(* CODESYS project Codesys

Project tree, tasks and I/O mapping:
  Device : PMCprimo Base, Pilz GmbH & Co. KG, version 3.5.15.1
    application Application
      libraries: Standard, 3.5.18.0 (System)
      task EtherCAT (externalevent, external event EVENT_ECM_DC, priority 0) calls EtherCAT_Master_Pilz.EtherCAT_Task, PLC_PRG
      task MainTask (cyclic, interval 1 ms, priority 0) calls nothing
      program PLC_PRG [LD]
    EtherCAT_Master_Pilz : EtherCAT_Master_Pilz, Pilz GmbH & Co. KG, version 3.5.17.0
        settings: NetworkName = 'ETHERCAT'; NetworkName = "ETHERCAT"; SrcAddress1 = 2; SrcAddress2 = 1212745857
      SI6_SC6_2Ax : SI6/SC6 2Ax, STOEBER ANTRIEBSTECHNIK GmbH & Co. KG, order no. SI6/SC6 2Ax, version Revision=16#00000011
          settings: ModularDevice = True; Number of Outputs = 0; Number of Inputs = 0; Number of Infos about Outputs = 0; Number of Infos about Inputs = 0; MDP_InputOffsets = [0,0,192]; MDP_OutputOffsets = [0,0,48]; Sync.Length = 12; Sync.Length = 44; FMMU.Length = 12; FMMU.Length = 44; Number of RxPDOs of the Slave = 2; Number of TxPDOs of the Slave = 2; DC sync0 cycletime = 1000; DC sync1 cycletime = 1000; RxTxPdo.NumberofExcludes = 0; RxTxPdo.NumberofEntries = 2; RxTxPdo.Index = 16#1600; RxTxPdo.Fixed = False; RxTxPdo.Mandatory = False; RxTxPdo.Virtual = False; RxTxPdo.Sm = 2; RxTxPdo.Su = 0; RxTxPdo.Name = 'Axis A to Slave'; RxTxPdo.DependOnSlot = False; RxTxPdo.DependOnSlotGroup = False; RxTxPdo.OverwrittenByModule = True; 1.A515 Controlword.Index = 16#6040; 1.A515 Controlword.SubIndex = 0; 1.A515 Controlword.Size = 16; 1.A515 Controlword.Offset = 0; 1.A515 Controlword.DependOnSlot = False; 1.A515 Controlword.DependOnSlotGroup = False; 1.A567 Target position.Index = 16#607A; 1.A567 Target position.SubIndex = 0; 1.A567 Target position.Size = 32; 1.A567 Target position.Offset = 0; 1.A567 Target position.DependOnSlot = False; 1.A567 Target position.DependOnSlotGroup = False; RxTxPdo.NumberofExcludes = 0;
            RxTxPdo.NumberofEntries = 2; RxTxPdo.Index = 16#1601; RxTxPdo.Fixed = False; RxTxPdo.Mandatory = False; RxTxPdo.Virtual = False; RxTxPdo.Sm = 2; RxTxPdo.Su = 0; RxTxPdo.Name = 'Axis B to Slave'; RxTxPdo.DependOnSlot = False; RxTxPdo.DependOnSlotGroup = False; RxTxPdo.OverwrittenByModule = True; 2.A515 Controlword.Index = 16#6840; 2.A515 Controlword.SubIndex = 0; 2.A515 Controlword.Size = 16; 2.A515 Controlword.Offset = 0; 2.A515 Controlword.DependOnSlot = False; 2.A515 Controlword.DependOnSlotGroup = False; 2.A567 Target position.Index = 16#687A; 2.A567 Target position.SubIndex = 0; 2.A567 Target position.Size = 32; 2.A567 Target position.Offset = 0; 2.A567 Target position.DependOnSlot = False; 2.A567 Target position.DependOnSlotGroup = False; RxTxPdo.NumberofExcludes = 0; RxTxPdo.NumberofEntries = 8; RxTxPdo.Index = 16#1A00; RxTxPdo.Fixed = False; RxTxPdo.Mandatory = False; RxTxPdo.Virtual = False; RxTxPdo.Sm = 3; RxTxPdo.Su = 0; RxTxPdo.Name = 'Axis A to Master'; RxTxPdo.DependOnSlot = False; RxTxPdo.DependOnSlotGroup = False; RxTxPdo.OverwrittenByModule = True; 1.A516 Statusword.Index = 16#6041; 1.A516 Statusword.SubIndex = 0; 1.A516 Statusword.Size = 16; 1.A516 Statusword.Offset = 0; 1.A516 Statusword.DependOnSlot = False;
            1.A516 Statusword.DependOnSlotGroup = False; 1.A545 Position actual value.Index = 16#6064; 1.A545 Position actual value.SubIndex = 0; 1.A545 Position actual value.Size = 32; 1.A545 Position actual value.Offset = 0; 1.A545 Position actual value.DependOnSlot = False; 1.A545 Position actual value.DependOnSlotGroup = False; 1.A564 Torque actual value.Index = 16#6077; 1.A564 Torque actual value.SubIndex = 0; 1.A564 Torque actual value.Size = 16; 1.A564 Torque actual value.Offset = 0; 1.A564 Torque actual value.DependOnSlot = False; 1.A564 Torque actual value.DependOnSlotGroup = False; 1.A636 Digital inputs.Index = 16#60FD; 1.A636 Digital inputs.SubIndex = 0; 1.A636 Digital inputs.Size = 32; 1.A636 Digital inputs.Offset = 0; 1.A636 Digital inputs.DependOnSlot = False; 1.A636 Digital inputs.DependOnSlotGroup = False; 1.A595 Touch probe status.Index = 16#60B9; 1.A595 Touch probe status.SubIndex = 0; 1.A595 Touch probe status.Size = 16; 1.A595 Touch probe status.Offset = 0; 1.A595 Touch probe status.DependOnSlot = False; 1.A595 Touch probe status.DependOnSlotGroup = False; 1.A596 Touch probe position 1 positive value.Index = 16#60BA; 1.A596 Touch probe position 1 positive value.SubIndex = 0; 1.A596 Touch probe position 1 positive value.Size = 32; 1.A596 Touch probe position 1 positive value.Offset = 0; 1.A596 Touch probe position 1 positive value.DependOnSlot = False; 1.A596 Touch probe position 1 positive value.DependOnSlotGroup = False; 1.A597 Touch probe position 1 negative value.Index = 16#60BB; 1.A597 Touch probe position 1 negative value.SubIndex = 0; 1.A597 Touch probe position 1 negative value.Size = 32; 1.A597 Touch probe position 1 negative value.Offset = 0; 1.A597 Touch probe position 1 negative value.DependOnSlot = False; 1.A597 Touch probe position 1 negative value.DependOnSlotGroup = False; 1.E201 Statuswort 2.Index = 16#28C9; 1.E201 Statuswort 2.SubIndex = 0; 1.E201 Statuswort 2.Size = 16;
            1.E201 Statuswort 2.Offset = 0; 1.E201 Statuswort 2.DependOnSlot = False; 1.E201 Statuswort 2.DependOnSlotGroup = False; RxTxPdo.NumberofExcludes = 0; RxTxPdo.NumberofEntries = 7; RxTxPdo.Index = 16#1A01; RxTxPdo.Fixed = False; RxTxPdo.Mandatory = False; RxTxPdo.Virtual = False; RxTxPdo.Sm = 3; RxTxPdo.Su = 0; RxTxPdo.Name = 'Axis B to Master'; RxTxPdo.DependOnSlot = False; RxTxPdo.DependOnSlotGroup = False; RxTxPdo.OverwrittenByModule = True; 2.A516 Statusword.Index = 16#6841; 2.A516 Statusword.SubIndex = 0; 2.A516 Statusword.Size = 16; 2.A516 Statusword.Offset = 0; 2.A516 Statusword.DependOnSlot = False; 2.A516 Statusword.DependOnSlotGroup = False; 2.A545 Position actual value.Index = 16#6864; 2.A545 Position actual value.SubIndex = 0; 2.A545 Position actual value.Size = 32; 2.A545 Position actual value.Offset = 0; 2.A545 Position actual value.DependOnSlot = False; 2.A545 Position actual value.DependOnSlotGroup = False; 2.A564 Torque actual value.Index = 16#6877; 2.A564 Torque actual value.SubIndex = 0; 2.A564 Torque actual value.Size = 16; 2.A564 Torque actual value.Offset = 0; 2.A564 Torque actual value.DependOnSlot = False; 2.A564 Torque actual value.DependOnSlotGroup = False; 2.A595 Touch probe status.Index = 16#68B9; 2.A595 Touch probe status.SubIndex = 0; 2.A595 Touch probe status.Size = 16; 2.A595 Touch probe status.Offset = 0; 2.A595 Touch probe status.DependOnSlot = False; 2.A595 Touch probe status.DependOnSlotGroup = False; 2.A596 Touch probe position 1 positive value.Index = 16#68BA;
            2.A596 Touch probe position 1 positive value.SubIndex = 0; 2.A596 Touch probe position 1 positive value.Size = 32; 2.A596 Touch probe position 1 positive value.Offset = 0; 2.A596 Touch probe position 1 positive value.DependOnSlot = False; 2.A596 Touch probe position 1 positive value.DependOnSlotGroup = False; 2.A597 Touch probe position 1 negative value.Index = 16#68BB; 2.A597 Touch probe position 1 negative value.SubIndex = 0; 2.A597 Touch probe position 1 negative value.Size = 32; 2.A597 Touch probe position 1 negative value.Offset = 0; 2.A597 Touch probe position 1 negative value.DependOnSlot = False; 2.A597 Touch probe position 1 negative value.DependOnSlotGroup = False; 1.E201 Statuswort 2.Index = 16#28C9; 1.E201 Statuswort 2.SubIndex = 0; 1.E201 Statuswort 2.Size = 16; 1.E201 Statuswort 2.Offset = 0; 1.E201 Statuswort 2.DependOnSlot = False; 1.E201 Statuswort 2.DependOnSlotGroup = False; 1.A515 Controlword.Name = '1.A515 Controlword'; 1.A515 Controlword.DataType = 'WORD'; 1.A515 Controlword.Default = ''; 1.A515 Controlword.Comment = ''; 1.A567 Target position.Name = '1.A567 Target position'; 1.A567 Target position.DataType = 'DINT'; 1.A567 Target position.Default = ''; 1.A567 Target position.Comment = ''; 2.A515 Controlword.Name = '2.A515 Controlword'; 2.A515 Controlword.DataType = 'WORD'; 2.A515 Controlword.Default = ''; 2.A515 Controlword.Comment = ''; 2.A567 Target position.Name = '2.A567 Target position'; 2.A567 Target position.DataType = 'DINT'; 2.A567 Target position.Default = ''; 2.A567 Target position.Comment = ''; 1.A516 Statusword.Name = '1.A516 Statusword'; 1.A516 Statusword.DataType = 'WORD'; 1.A516 Statusword.Default = ''; 1.A516 Statusword.Comment = ''; 1.A545 Position actual value.Name = '1.A545 Position actual value'; 1.A545 Position actual value.DataType = 'DINT'; 1.A545 Position actual value.Default = '';
            1.A545 Position actual value.Comment = ''; 1.A564 Torque actual value.Name = '1.A564 Torque actual value'; 1.A564 Torque actual value.DataType = 'INT'; 1.A564 Torque actual value.Default = ''; 1.A564 Torque actual value.Comment = ''; 1.A636 Digital inputs.Name = '1.A636 Digital inputs'; 1.A636 Digital inputs.DataType = 'DWORD'; 1.A636 Digital inputs.Default = ''; 1.A636 Digital inputs.Comment = ''; 1.A595 Touch probe status.Name = '1.A595 Touch probe status'; 1.A595 Touch probe status.DataType = 'WORD'; 1.A595 Touch probe status.Default = ''; 1.A595 Touch probe status.Comment = ''; 1.A596 Touch probe position 1 positive value.Name = '1.A596 Touch probe position 1 positive value'; 1.A596 Touch probe position 1 positive value.DataType = 'DINT'; 1.A596 Touch probe position 1 positive value.Default = ''; 1.A596 Touch probe position 1 positive value.Comment = ''; 1.A597 Touch probe position 1 negative value.Name = '1.A597 Touch probe position 1 negative value'; 1.A597 Touch probe position 1 negative value.DataType = 'DINT'; 1.A597 Touch probe position 1 negative value.Default = ''; 1.A597 Touch probe position 1 negative value.Comment = ''; 1.E201 Statuswort 2.Name = '1.E201 Statuswort 2'; 1.E201 Statuswort 2.DataType = 'WORD'; 1.E201 Statuswort 2.Default = ''; 1.E201 Statuswort 2.Comment = ''; 2.A516 Statusword.Name = '2.A516 Statusword'; 2.A516 Statusword.DataType = 'WORD'; 2.A516 Statusword.Default = ''; 2.A516 Statusword.Comment = ''; 2.A545 Position actual value.Name = '2.A545 Position actual value'; 2.A545 Position actual value.DataType = 'DINT'; 2.A545 Position actual value.Default = ''; 2.A545 Position actual value.Comment = ''; 2.A564 Torque actual value.Name = '2.A564 Torque actual value'; 2.A564 Torque actual value.DataType = 'INT'; 2.A564 Torque actual value.Default = ''; 2.A564 Torque actual value.Comment = ''; 2.A595 Touch probe status.Name = '2.A595 Touch probe status'; 2.A595 Touch probe status.DataType = 'WORD'; 2.A595 Touch probe status.Default = '';
            2.A595 Touch probe status.Comment = ''; 2.A596 Touch probe position 1 positive value.Name = '2.A596 Touch probe position 1 positive value'; 2.A596 Touch probe position 1 positive value.DataType = 'DINT'; 2.A596 Touch probe position 1 positive value.Default = ''; 2.A596 Touch probe position 1 positive value.Comment = ''; 2.A597 Touch probe position 1 negative value.Name = '2.A597 Touch probe position 1 negative value'; 2.A597 Touch probe position 1 negative value.DataType = 'DINT'; 2.A597 Touch probe position 1 negative value.Default = ''; 2.A597 Touch probe position 1 negative value.Comment = ''; 1.E201 Statuswort 2.Name = '1.E201 Statuswort 2'; 1.E201 Statuswort 2.DataType = 'WORD'; 1.E201 Statuswort 2.Default = ''; 1.E201 Statuswort 2.Comment = ''
        Axis_A : xA PMCprimo-SI6/SC6_0, STOEBER ANTRIEBSTECHNIK GmbH & Co. KG, order no. PMCprimo-SI6/SC6_0, version 0
            settings: Number of Outputs = 2; Number of Inputs = 8; Number of Infos about Outputs = 2; Number of Infos about Inputs = 8; RxTxPdo.Mandatory = False; RxTxPdo.Virtual = False; RxTxPdo.DependOnSlot = False; RxTxPdo.DependOnSlotGroup = False; RxTxPdo.OverwrittenByModule = True; 1.A515 Controlword.Offset = 0; 1.A515 Controlword.DependOnSlot = False; 1.A515 Controlword.DependOnSlotGroup = False; 1.A567 Target position.Offset = 0; 1.A567 Target position.DependOnSlot = False; 1.A567 Target position.DependOnSlotGroup = False; RxTxPdo.Mandatory = False; RxTxPdo.Virtual = False; RxTxPdo.DependOnSlot = False; RxTxPdo.DependOnSlotGroup = False; RxTxPdo.OverwrittenByModule = True; 1.A516 Statusword.Offset = 0; 1.A516 Statusword.DependOnSlot = False; 1.A516 Statusword.DependOnSlotGroup = False; 1.A545 Position actual value.Offset = 0; 1.A545 Position actual value.DependOnSlot = False; 1.A545 Position actual value.DependOnSlotGroup = False; 1.A564 Torque actual value.Offset = 0; 1.A564 Torque actual value.DependOnSlot = False; 1.A564 Torque actual value.DependOnSlotGroup = False; 1.A636 Digital inputs.Offset = 0; 1.A636 Digital inputs.DependOnSlot = False; 1.A636 Digital inputs.DependOnSlotGroup = False; 1.A595 Touch probe status.Offset = 0; 1.A595 Touch probe status.DependOnSlot = False; 1.A595 Touch probe status.DependOnSlotGroup = False; 1.A596 Touch probe position 1 positive value.Offset = 0; 1.A596 Touch probe position 1 positive value.DependOnSlot = False; 1.A596 Touch probe position 1 positive value.DependOnSlotGroup = False; 1.A597 Touch probe position 1 negative value.Offset = 0; 1.A597 Touch probe position 1 negative value.DependOnSlot = False;
              1.A597 Touch probe position 1 negative value.DependOnSlotGroup = False; 1.E201 Statuswort 2.Offset = 0; 1.E201 Statuswort 2.DependOnSlot = False; 1.E201 Statuswort 2.DependOnSlotGroup = False; 1.A515 Controlword.Default = ''; 1.A567 Target position.Default = ''; 1.A516 Statusword.Default = ''; 1.A545 Position actual value.Default = ''; 1.A564 Torque actual value.Default = ''; 1.A636 Digital inputs.Default = ''; 1.A595 Touch probe status.Default = ''; 1.A596 Touch probe position 1 positive value.Default = ''; 1.A597 Touch probe position 1 negative value.Default = ''; 1.E201 Statuswort 2.Default = ''
            unmapped channels: 1.A515 Controlword, 1.A567 Target position, 1.A516 Statusword, 1.A545 Position actual value, 1.A564 Torque actual value, 1.A636 Digital inputs, 1.A595 Touch probe status, 1.A596 Touch probe position 1 positive value, 1.A597 Touch probe position 1 negative value, 1.E201 Statuswort 2
        Axis_B : xB PMCprimo-SI6/SC6_1, STOEBER ANTRIEBSTECHNIK GmbH & Co. KG, order no. PMC-SI6/SC6_1, version 0
            settings: Number of Outputs = 2; Number of Inputs = 7; Number of Infos about Outputs = 2; Number of Infos about Inputs = 7; RxTxPdo.Mandatory = False; RxTxPdo.Virtual = False; RxTxPdo.DependOnSlot = False; RxTxPdo.DependOnSlotGroup = False; RxTxPdo.OverwrittenByModule = True; 2.A515 Controlword.Offset = 0; 2.A515 Controlword.DependOnSlot = False; 2.A515 Controlword.DependOnSlotGroup = False; 2.A567 Target position.Offset = 0; 2.A567 Target position.DependOnSlot = False; 2.A567 Target position.DependOnSlotGroup = False; RxTxPdo.Mandatory = False; RxTxPdo.Virtual = False; RxTxPdo.DependOnSlot = False; RxTxPdo.DependOnSlotGroup = False; RxTxPdo.OverwrittenByModule = True; 2.A516 Statusword.Offset = 0; 2.A516 Statusword.DependOnSlot = False; 2.A516 Statusword.DependOnSlotGroup = False; 2.A545 Position actual value.Offset = 0; 2.A545 Position actual value.DependOnSlot = False; 2.A545 Position actual value.DependOnSlotGroup = False; 2.A564 Torque actual value.Offset = 0; 2.A564 Torque actual value.DependOnSlot = False; 2.A564 Torque actual value.DependOnSlotGroup = False; 2.A595 Touch probe status.Offset = 0; 2.A595 Touch probe status.DependOnSlot = False; 2.A595 Touch probe status.DependOnSlotGroup = False; 2.A596 Touch probe position 1 positive value.Offset = 0; 2.A596 Touch probe position 1 positive value.DependOnSlot = False; 2.A596 Touch probe position 1 positive value.DependOnSlotGroup = False; 2.A597 Touch probe position 1 negative value.Offset = 0; 2.A597 Touch probe position 1 negative value.DependOnSlot = False; 2.A597 Touch probe position 1 negative value.DependOnSlotGroup = False; 1.E201 Statuswort 2.Offset = 0; 1.E201 Statuswort 2.DependOnSlot = False;
              1.E201 Statuswort 2.DependOnSlotGroup = False; 2.A515 Controlword.Default = ''; 2.A567 Target position.Default = ''; 2.A516 Statusword.Default = ''; 2.A545 Position actual value.Default = ''; 2.A564 Torque actual value.Default = ''; 2.A595 Touch probe status.Default = ''; 2.A596 Touch probe position 1 positive value.Default = ''; 2.A597 Touch probe position 1 negative value.Default = ''; 1.E201 Statuswort 2.Default = ''
            unmapped channels: 2.A515 Controlword, 2.A567 Target position, 2.A516 Statusword, 2.A545 Position actual value, 2.A564 Torque actual value, 2.A595 Touch probe status, 2.A596 Touch probe position 1 positive value, 2.A597 Touch probe position 1 negative value, 1.E201 Statuswort 2
  program POU [ST]
*)

// Device/Application/PLC_PRG
PROGRAM PLC_PRG
VAR
	InterfaceEtherCAT_: primoCE_C3.PrimoEtherCATInterface;
END_VAR

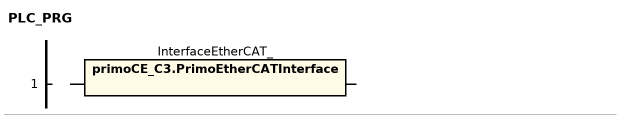
// NETWORK 1
InterfaceEtherCAT_(); // primoCE_C3.PrimoEtherCATInterface

END_PROGRAM

// POU
PROGRAM POU
VAR
	Fabien:BOOL;
	Bobby:bool;
END_VAR

END_PROGRAM
